{attribute 'pack_mode' := '2'}
TYPE ST_STATION_STATE :
STRUCT
  State           : E_STATION_STATE;
  {attribute 'displaymode':='bin'}
  nMask           : BYTE;
  nMoverId        : USINT;
  rMoverModPos    : LREAL;            // modulo position of detected mover
  nQueue          : USINT;            // queue count for station
END_STRUCT
END_TYPE

(* stored: Version 1.1.0.1, ProductVersion 3.1.4026.18
   DUT ST_STATION_STATE: Id {d36cc9f2-a002-4877-832c-78f9675b049f} *)
